% RSLogix 500 project LAB 10 Stop Light TON.RSS %
PROJECT "UNTITLED"    % processor: MicroLogix 1500 %

PROGRAM FILES
  LAD 2   11 rungs

DATA FILES
  O0 OUTPUT  4 elements
  I1 INPUT  4 elements
  S2 STATUS  66 elements
  B3 BINARY  1 elements
  T4 TIMER  5 elements
  C5 COUNTER  1 elements
  R6 CONTROL  1 elements
  N7 INTEGER  1 elements
  F8 FLOAT  1 elements

LADDER 2
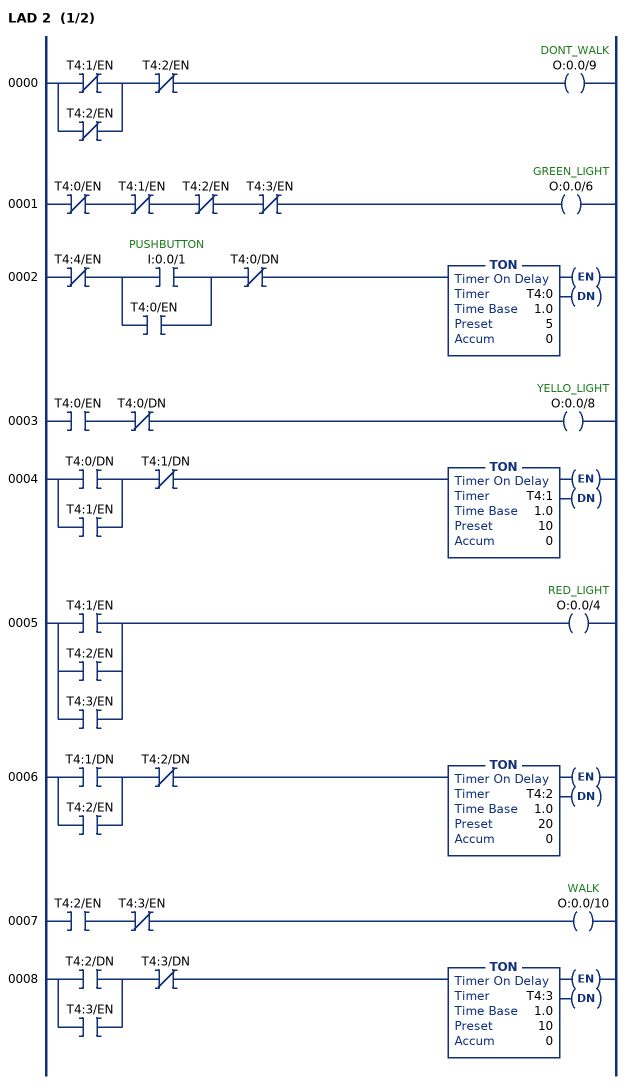
% Rung: 0 %
SOR BST XIO T4:1/EN NXB XIO T4:2/EN BND XIO T4:2/EN OTE O:0.0/9 EOR
%   O:0.0/9  DONT_WALK %
% Rung: 1 %
SOR XIO T4:0/EN XIO T4:1/EN XIO T4:2/EN XIO T4:3/EN OTE O:0.0/6 EOR
%   O:0.0/6  GREEN_LIGHT %
% Rung: 2 %
SOR XIO T4:4/EN BST XIC I:0.0/1 NXB XIC T4:0/EN BND XIO T4:0/DN TON T4:0 1.0 5 0 EOR
%   I:0.0/1  PUSHBUTTON %
% Rung: 3 %
SOR XIC T4:0/EN XIO T4:0/DN OTE O:0.0/8 EOR
%   O:0.0/8  YELLO_LIGHT %
% Rung: 4 %
SOR BST XIC T4:0/DN NXB XIC T4:1/EN BND XIO T4:1/DN TON T4:1 1.0 10 0 EOR
% Rung: 5 %
SOR BST BST XIC T4:1/EN NXB XIC T4:2/EN BND NXB XIC T4:3/EN BND OTE O:0.0/4 EOR
%   O:0.0/4  RED_LIGHT %
% Rung: 6 %
SOR BST XIC T4:1/DN NXB XIC T4:2/EN BND XIO T4:2/DN TON T4:2 1.0 20 0 EOR
% Rung: 7 %
SOR XIC T4:2/EN XIO T4:3/EN OTE O:0.0/10 EOR
%   O:0.0/10  WALK %
% Rung: 8 %
SOR BST XIC T4:2/DN NXB XIC T4:3/EN BND XIO T4:3/DN TON T4:3 1.0 10 0 EOR

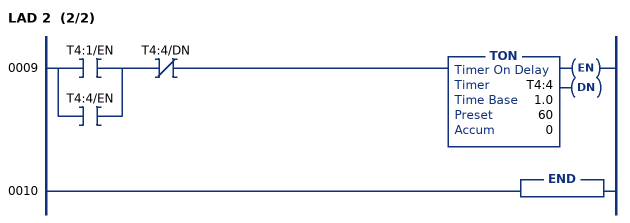
% Rung: 9 %
SOR BST XIC T4:1/EN NXB XIC T4:4/EN BND XIO T4:4/DN TON T4:4 1.0 60 0 EOR
% Rung: 10 %
SOR END EOR

OTHER DOCUMENTED ADDRESSES
  I:0.0/0  ZERO
  O:0.0/0  OUT_ZERO
  O:0.0/1  ONE
  O:0.0/2  TWO
  O:0.0/3  THREE

DATA TABLE (non-zero values as saved)
DATA T4
% .PRE .ACC %
% T4:0 % 5 0
% T4:1 % 10 0
% T4:2 % 20 0
% T4:3 % 10 0
% T4:4 % 60 0
